(* Schneider Machine Expert - Basic project New project, file version 1.6.0.0 *)
(* ProjectInformations: Name=New project *)

HARDWARE
  Cpu 0: TM221CE16R
  EthernetConfiguration: NetworkName=M221, IpAllocationMode=FixedAddress, IpAddress=0.0.0.0, SubnetMask=0.0.0.0
  SerialLineConfiguration: Baud=Baud19200, Parity=ParityEven, DataBits=DataBits8, StopBits=StopBits1, PhysicalMedium=PhysicalMediumRs485, TransmissionMode=TransmissionModeModbusRtu, SlaveId=1, Addressing=SlaveAddressing
  MastTask: UsePeriodScanMode=false, PeriodScan=100
  FastTask: Period=255
  CpuBehavior: StartingMode=StartAsPreviousState, AutoSaveRamOnEeprom=true, WatchdogPeriod=250

SYMBOLS  (address, symbol, comment, settings)
  %TM0        [Preset=1211, Base=OneSecond]

POU New POU
  (* SectionNumber=1 *)

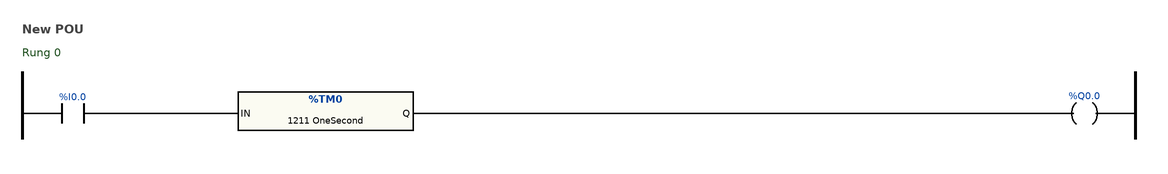

// Rung 0
  BLK %TM0
  LD %I0.0
  IN
  OUT_BLK
  LD Q
  ST %Q0.0
  END_BLK
  // as ST:
  //   %TM0(IN := %I0.0);
  //   %Q0.0 := %TM0.Q;
